Fanuc KAREL source: kd00017.KL

-- PROVISIONAL review KL for V770-1; original PC SHA256 8bccabb68298124adb2e00a3fafcbc7a19fd06749926fa88ddc8507115944daa
-- Incomplete behavior may be omitted. Consult companion uncertainty JSON. Do not deploy.
PROGRAM KD00017
%NOLOCKGROUP
VAR
  I : INTEGER
  J : INTEGER
  B : BOOLEAN
  R : REAL
  S : STRING[80]
BEGIN
  -- UNRESOLVED_PC offsets 5-12; opcodes 9C,23
  -- UNRESOLVED_PC offsets 17-24; opcodes 22,62
  -- UNRESOLVED_PC offsets 29-36; opcodes 22,28
  -- UNRESOLVED_PC offsets 41-45; opcodes 7F
END KD00017
